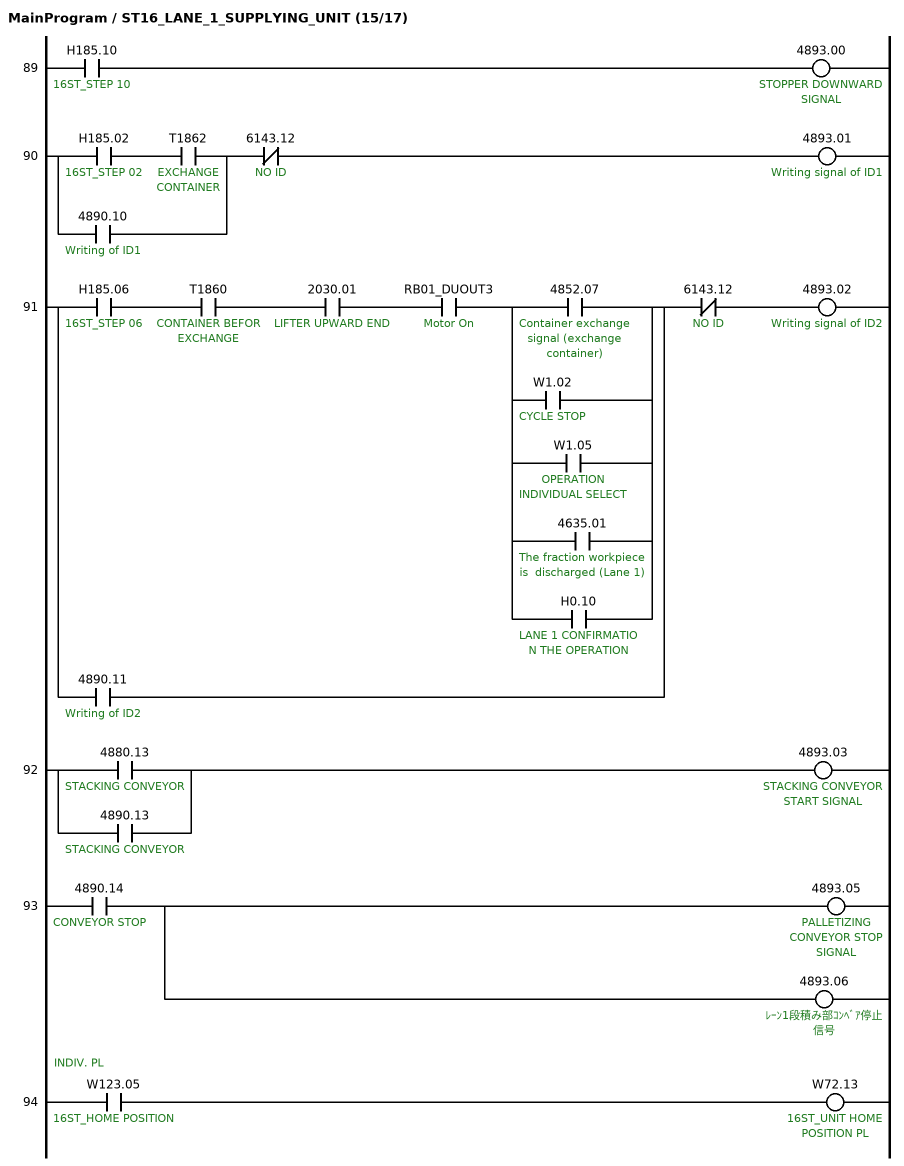
; [picture p648: MainProgram / ST16_LANE_1_SUPPLYING_UNIT, rungs 89-94]
; rung 89
LD H185.10  ; 16ST_STEP 10
OUT 4893.00  ; STOPPER DOWNWARD SIGNAL
; rung 90
LD H185.02  ; 16ST_STEP 02
AND T1862  ; EXCHANGE CONTAINER
OR 4890.10  ; Writing of ID1
ANDNOT 6143.12  ; NO ID
OUT 4893.01  ; Writing signal of ID1
; rung 91
LD H185.06  ; 16ST_STEP 06
AND T1860  ; CONTAINER BEFOR EXCHANGE
AND 2030.01  ; LIFTER UPWARD END
AND RB01_DUOUT3  ; Motor On
LD 4852.07  ; Container exchange signal (exchange container)
OR W1.02  ; CYCLE STOP
OR W1.05  ; OPERATION INDIVIDUAL SELECT
OR 4635.01  ; The fraction workpiece is  discharged (Lane 1)
OR H0.10  ; LANE 1 CONFIRMATION THE OPERATION
ANDLD
OR 4890.11  ; Writing of ID2
ANDNOT 6143.12  ; NO ID
OUT 4893.02  ; Writing signal of ID2
; rung 92
LD 4880.13  ; STACKING CONVEYOR
OR 4890.13  ; STACKING CONVEYOR
OUT 4893.03  ; STACKING CONVEYOR START SIGNAL
; rung 93
LD 4890.14  ; CONVEYOR STOP
OUT 4893.05  ; PALLETIZING CONVEYOR STOP SIGNAL
OUT 4893.06  ; ﾚｰﾝ1段積み部ｺﾝﾍﾞｱ停止信号
; rung 94: INDIV. PL
LD W123.05  ; 16ST_HOME POSITION
OUT W72.13  ; 16ST_UNIT HOME POSITION PL

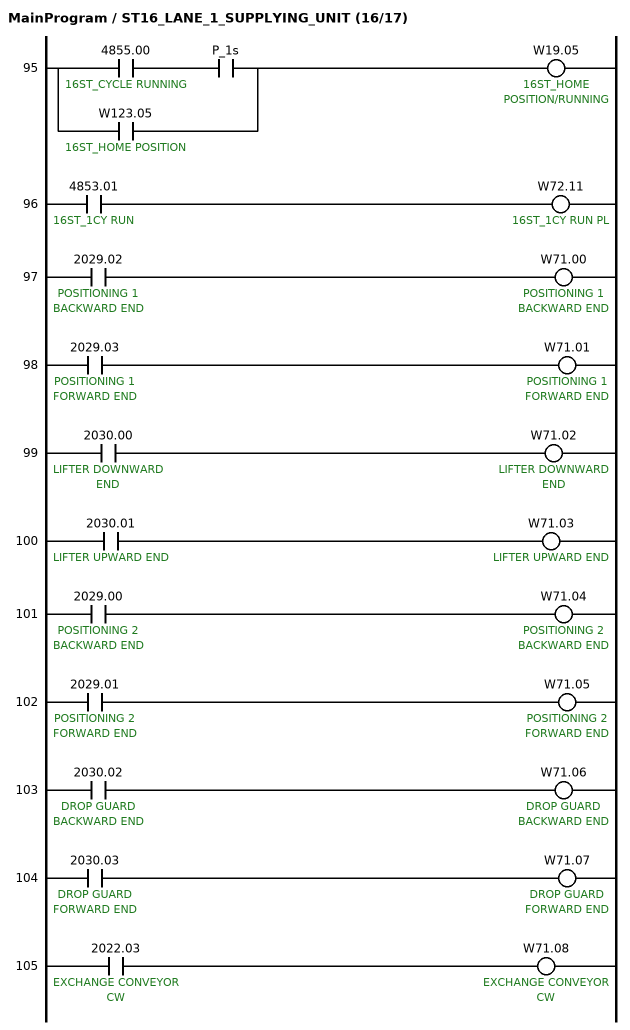
; rung 95
LD 4855.00  ; 16ST_CYCLE RUNNING
AND P_1s
OR W123.05  ; 16ST_HOME POSITION
OUT W19.05  ; 16ST_HOME POSITION/RUNNING
; rung 96
LD 4853.01  ; 16ST_1CY RUN
OUT W72.11  ; 16ST_1CY RUN PL
; rung 97
LD 2029.02  ; POSITIONING 1 BACKWARD END
OUT W71.00  ; POSITIONING 1 BACKWARD END
; rung 98
LD 2029.03  ; POSITIONING 1 FORWARD END
OUT W71.01  ; POSITIONING 1 FORWARD END
; rung 99
LD 2030.00  ; LIFTER DOWNWARD END
OUT W71.02  ; LIFTER DOWNWARD END
; rung 100
LD 2030.01  ; LIFTER UPWARD END
OUT W71.03  ; LIFTER UPWARD END
; rung 101
LD 2029.00  ; POSITIONING 2 BACKWARD END
OUT W71.04  ; POSITIONING 2 BACKWARD END
; rung 102
LD 2029.01  ; POSITIONING 2 FORWARD END
OUT W71.05  ; POSITIONING 2 FORWARD END
; rung 103
LD 2030.02  ; DROP GUARD BACKWARD END
OUT W71.06  ; DROP GUARD BACKWARD END
; rung 104
LD 2030.03  ; DROP GUARD FORWARD END
OUT W71.07  ; DROP GUARD FORWARD END
; rung 105
LD 2022.03  ; EXCHANGE CONVEYOR CW
OUT W71.08  ; EXCHANGE CONVEYOR CW

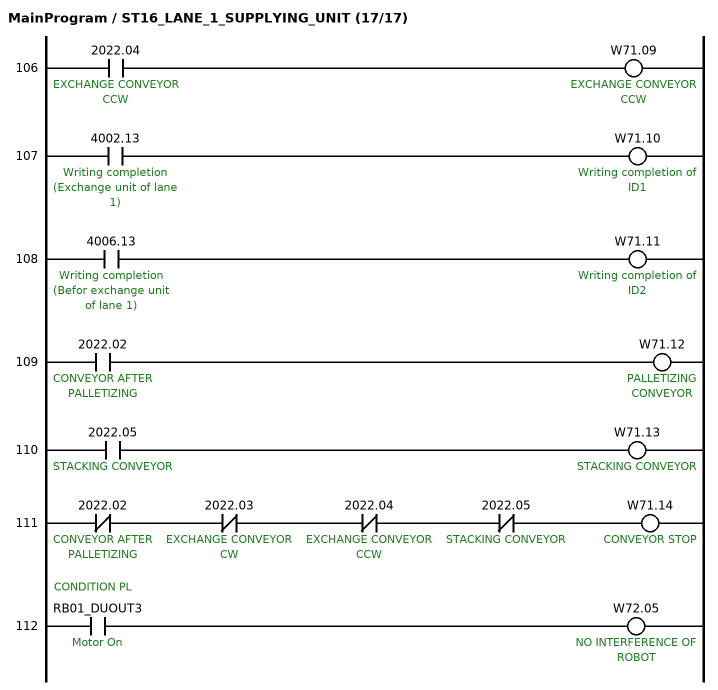
; rung 106
LD 2022.04  ; EXCHANGE CONVEYOR CCW
OUT W71.09  ; EXCHANGE CONVEYOR CCW
; rung 107
LD 4002.13  ; Writing completion (Exchange unit of lane 1)
OUT W71.10  ; Writing completion of ID1
; rung 108
LD 4006.13  ; Writing completion (Befor exchange unit of lane 1)
OUT W71.11  ; Writing completion of ID2
; rung 109
LD 2022.02  ; CONVEYOR AFTER PALLETIZING
OUT W71.12  ; PALLETIZING CONVEYOR
; rung 110
LD 2022.05  ; STACKING CONVEYOR
OUT W71.13  ; STACKING CONVEYOR
; rung 111
LDNOT 2022.02  ; CONVEYOR AFTER PALLETIZING
ANDNOT 2022.03  ; EXCHANGE CONVEYOR CW
ANDNOT 2022.04  ; EXCHANGE CONVEYOR CCW
ANDNOT 2022.05  ; STACKING CONVEYOR
OUT W71.14  ; CONVEYOR STOP
; rung 112: CONDITION PL
LD RB01_DUOUT3  ; Motor On
OUT W72.05  ; NO INTERFERENCE OF ROBOT

### Section ST17_LANE_1_STACKING_UNIT

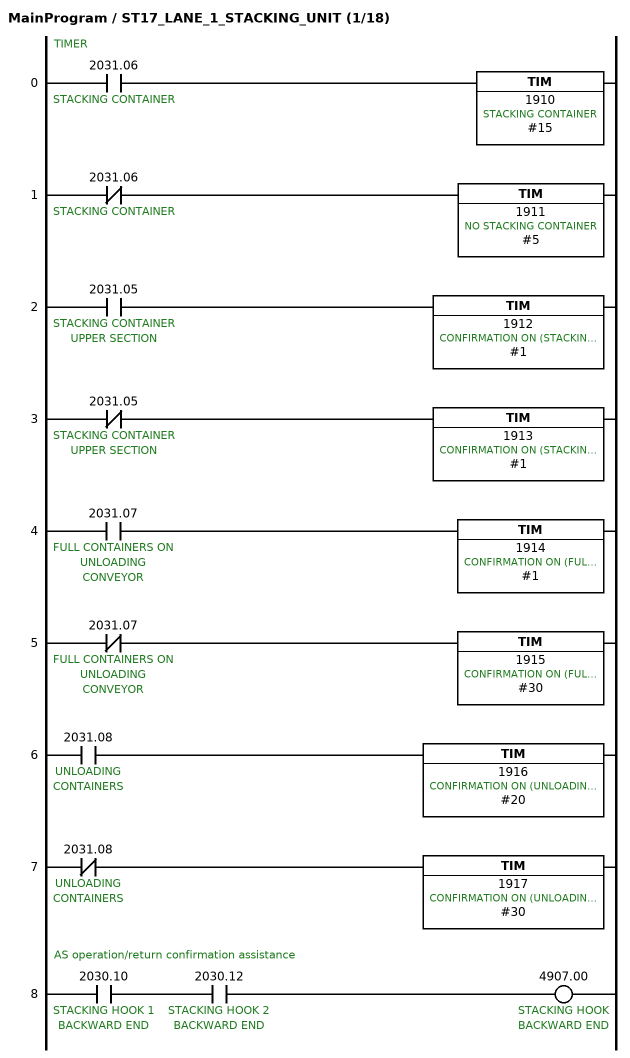
; rung 0: TIMER
LD 2031.06  ; STACKING CONTAINER
TIM 1910 #15  ; STACKING CONTAINER
; rung 1
LDNOT 2031.06  ; STACKING CONTAINER
TIM 1911 #5  ; NO STACKING CONTAINER
; rung 2
LD 2031.05  ; STACKING CONTAINER UPPER SECTION
TIM 1912 #1  ; CONFIRMATION ON (STACKING CONTAINER UPPER SECTION)
; rung 3
LDNOT 2031.05  ; STACKING CONTAINER UPPER SECTION
TIM 1913 #1  ; CONFIRMATION ON (STACKING CONTAINER UPPER SECTION)
; rung 4
LD 2031.07  ; FULL CONTAINERS ON UNLOADING CONVEYOR
TIM 1914 #1  ; CONFIRMATION ON (FULL CONTAINERS ON UNLOADING CONVEYOR)
; rung 5
LDNOT 2031.07  ; FULL CONTAINERS ON UNLOADING CONVEYOR
TIM 1915 #30  ; CONFIRMATION ON (FULL CONTAINERS ON UNLOADING CONVEYOR)
; rung 6
LD 2031.08  ; UNLOADING CONTAINERS
TIM 1916 #20  ; CONFIRMATION ON (UNLOADING CONTAINERS)
; rung 7
LDNOT 2031.08  ; UNLOADING CONTAINERS
TIM 1917 #30  ; CONFIRMATION ON (UNLOADING CONTAINERS)
; rung 8: AS operation/return confirmation assistance
LD 2030.10  ; STACKING HOOK 1 BACKWARD END
AND 2030.12  ; STACKING HOOK 2 BACKWARD END
OUT 4907.00  ; STACKING HOOK BACKWARD END

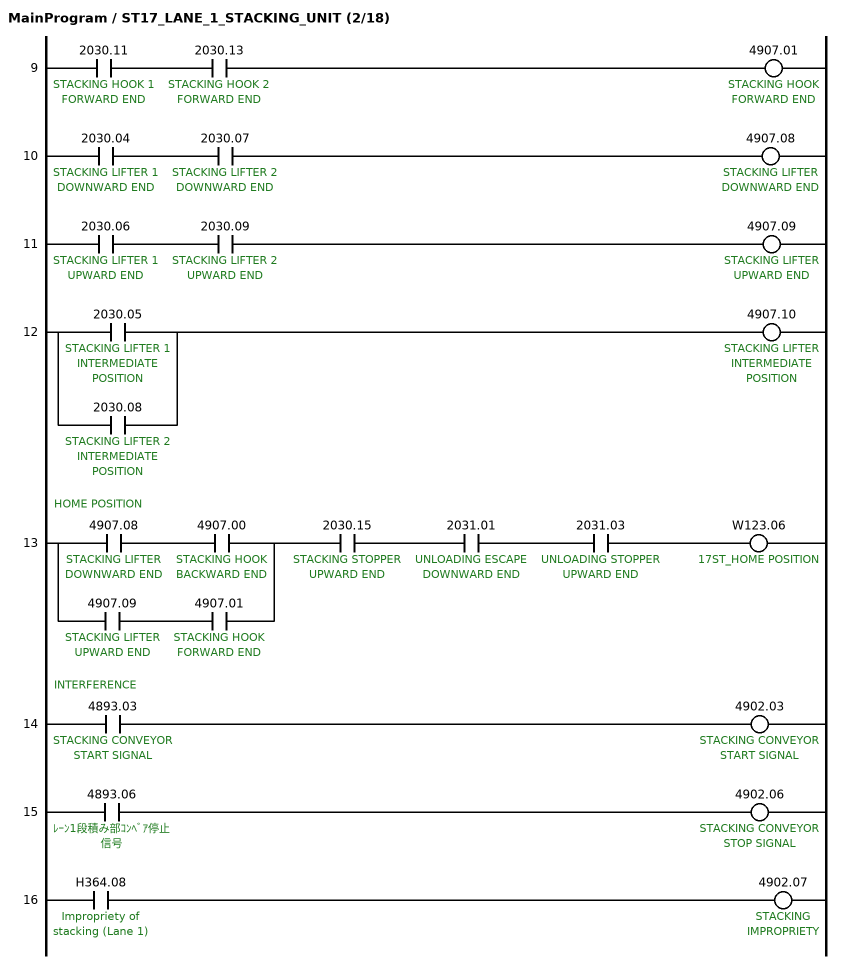
; rung 9
LD 2030.11  ; STACKING HOOK 1 FORWARD END
AND 2030.13  ; STACKING HOOK 2 FORWARD END
OUT 4907.01  ; STACKING HOOK FORWARD END
; rung 10
LD 2030.04  ; STACKING LIFTER 1 DOWNWARD END
AND 2030.07  ; STACKING LIFTER 2 DOWNWARD END
OUT 4907.08  ; STACKING LIFTER DOWNWARD END
; rung 11
LD 2030.06  ; STACKING LIFTER 1 UPWARD END
AND 2030.09  ; STACKING LIFTER 2 UPWARD END
OUT 4907.09  ; STACKING LIFTER UPWARD END
; rung 12
LD 2030.05  ; STACKING LIFTER 1 INTERMEDIATE POSITION
OR 2030.08  ; STACKING LIFTER 2 INTERMEDIATE POSITION
OUT 4907.10  ; STACKING LIFTER INTERMEDIATE POSITION
; rung 13: HOME POSITION
LD 4907.08  ; STACKING LIFTER DOWNWARD END
AND 4907.00  ; STACKING HOOK BACKWARD END
LD 4907.09  ; STACKING LIFTER UPWARD END
AND 4907.01  ; STACKING HOOK FORWARD END
ORLD
AND 2030.15  ; STACKING STOPPER UPWARD END
AND 2031.01  ; UNLOADING ESCAPE DOWNWARD END
AND 2031.03  ; UNLOADING STOPPER UPWARD END
OUT W123.06  ; 17ST_HOME POSITION
; rung 14: INTERFERENCE
LD 4893.03  ; STACKING CONVEYOR START SIGNAL
OUT 4902.03  ; STACKING CONVEYOR START SIGNAL
; rung 15
LD 4893.06  ; ﾚｰﾝ1段積み部ｺﾝﾍﾞｱ停止信号
OUT 4902.06  ; STACKING CONVEYOR STOP SIGNAL
; rung 16
LD H364.08  ; Impropriety of stacking (Lane 1)
OUT 4902.07  ; STACKING IMPROPRIETY

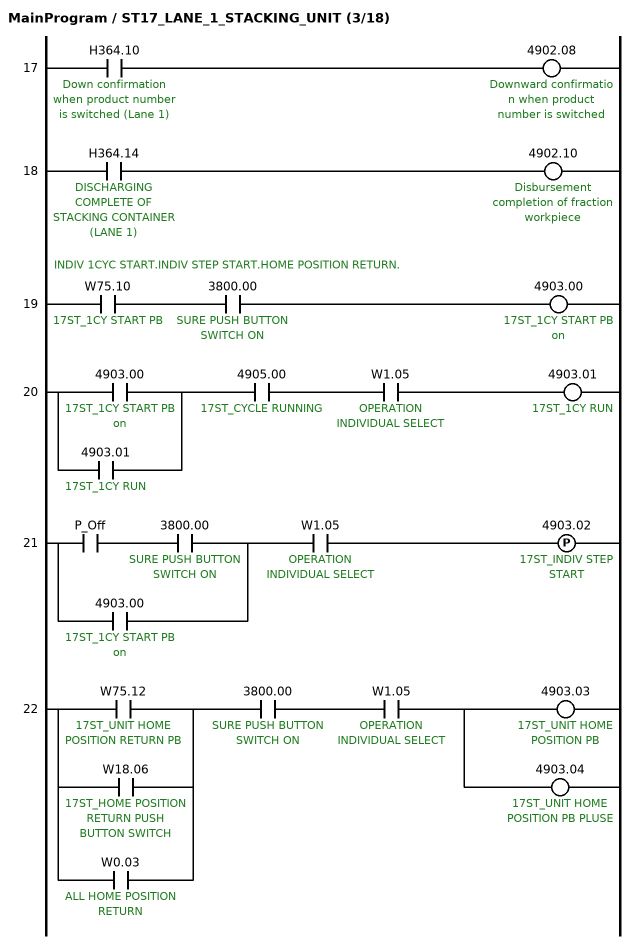
; rung 17
LD H364.10  ; Down confirmation when product number is switched (Lane 1)
OUT 4902.08  ; Downward confirmation when product number is switched
; rung 18
LD H364.14  ; DISCHARGING COMPLETE OF STACKING CONTAINER  (LANE 1)
OUT 4902.10  ; Disbursement completion of fraction workpiece
; rung 19: INDIV 1CYC START.INDIV STEP START.HOME POSITION RETURN.
LD W75.10  ; 17ST_1CY START PB
AND 3800.00  ; SURE PUSH BUTTON SWITCH ON
OUT 4903.00  ; 17ST_1CY START PB on
; rung 20
LD 4903.00  ; 17ST_1CY START PB on
OR 4903.01  ; 17ST_1CY RUN
AND 4905.00  ; 17ST_CYCLE RUNNING
AND W1.05  ; OPERATION INDIVIDUAL SELECT
OUT 4903.01  ; 17ST_1CY RUN
; rung 21
LD P_Off
AND 3800.00  ; SURE PUSH BUTTON SWITCH ON
OR 4903.00  ; 17ST_1CY START PB on
AND W1.05  ; OPERATION INDIVIDUAL SELECT
DIFU(013) 4903.02  ; 17ST_INDIV STEP START
; rung 22
LD W75.12  ; 17ST_UNIT HOME POSITION RETURN PB
OR W18.06  ; 17ST_HOME POSITION RETURN PUSH BUTTON SWITCH
OR W0.03  ; ALL HOME POSITION RETURN
AND 3800.00  ; SURE PUSH BUTTON SWITCH ON
AND W1.05  ; OPERATION INDIVIDUAL SELECT
OUT 4903.03  ; 17ST_UNIT HOME POSITION PB
OUT 4903.04  ; 17ST_UNIT HOME POSITION PB PLUSE

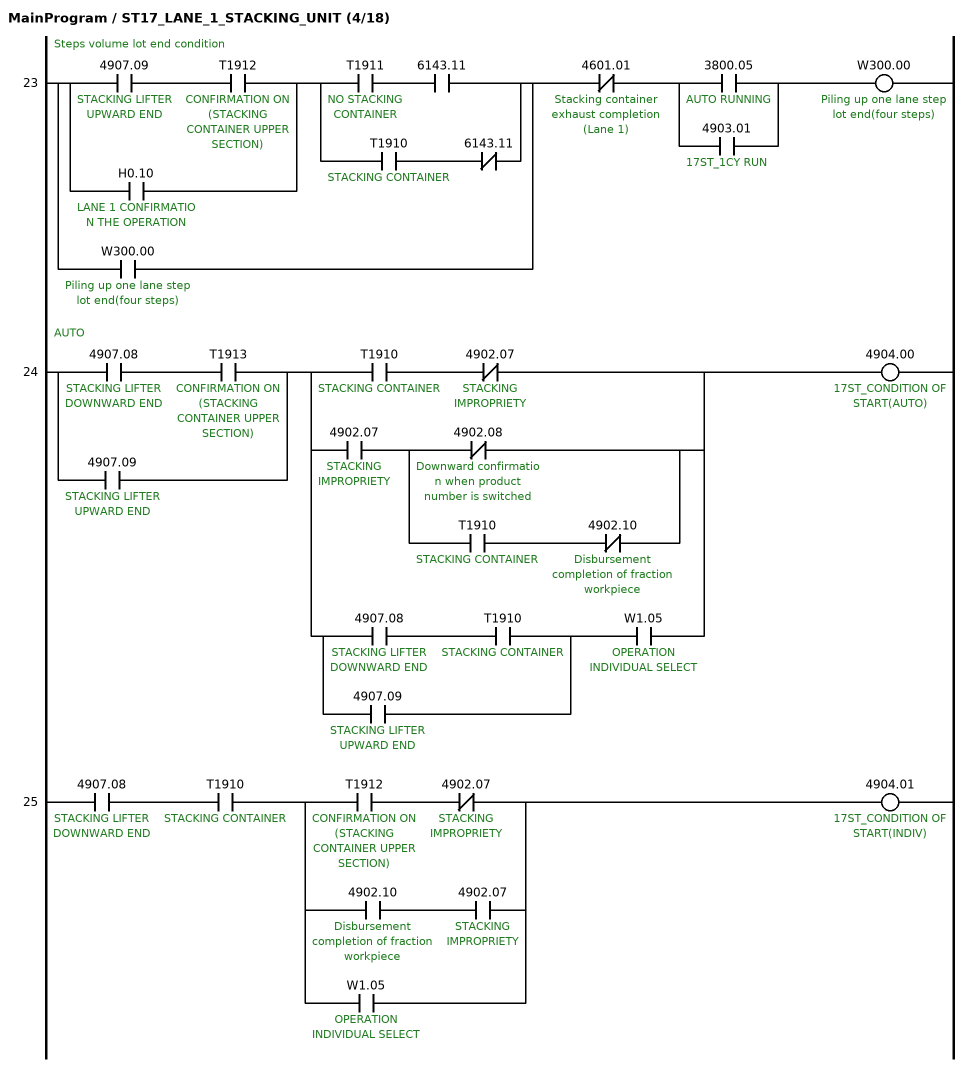
; rung 23: Steps volume lot end condition
LD 4907.09  ; STACKING LIFTER UPWARD END
AND T1912  ; CONFIRMATION ON (STACKING CONTAINER UPPER SECTION)
OR H0.10  ; LANE 1 CONFIRMATION THE OPERATION
LD T1911  ; NO STACKING CONTAINER
AND 6143.11
LD T1910  ; STACKING CONTAINER
ANDNOT 6143.11
ORLD
ANDLD
OR W300.00  ; Piling up one lane step lot end(four steps)
ANDNOT 4601.01  ; Stacking container exhaust completion (Lane 1)
LD 3800.05  ; AUTO RUNNING
OR 4903.01  ; 17ST_1CY RUN
ANDLD
OUT W300.00  ; Piling up one lane step lot end(four steps)
; rung 24: AUTO
LD 4907.08  ; STACKING LIFTER DOWNWARD END
AND T1913  ; CONFIRMATION ON (STACKING CONTAINER UPPER SECTION)
OR 4907.09  ; STACKING LIFTER UPWARD END
LD T1910  ; STACKING CONTAINER
ANDNOT 4902.07  ; STACKING IMPROPRIETY
LD 4902.07  ; STACKING IMPROPRIETY
LDNOT 4902.08  ; Downward confirmation when product number is switched
LD T1910  ; STACKING CONTAINER
ANDNOT 4902.10  ; Disbursement completion of fraction workpiece
ORLD
ANDLD
ORLD
LD 4907.08  ; STACKING LIFTER DOWNWARD END
AND T1910  ; STACKING CONTAINER
OR 4907.09  ; STACKING LIFTER UPWARD END
AND W1.05  ; OPERATION INDIVIDUAL SELECT
ORLD
ANDLD
OUT 4904.00  ; 17ST_CONDITION OF START(AUTO)
; rung 25
LD 4907.08  ; STACKING LIFTER DOWNWARD END
AND T1910  ; STACKING CONTAINER
LD T1912  ; CONFIRMATION ON (STACKING CONTAINER UPPER SECTION)
ANDNOT 4902.07  ; STACKING IMPROPRIETY
LD 4902.10  ; Disbursement completion of fraction workpiece
AND 4902.07  ; STACKING IMPROPRIETY
ORLD
OR W1.05  ; OPERATION INDIVIDUAL SELECT
ANDLD
OUT 4904.01  ; 17ST_CONDITION OF START(INDIV)

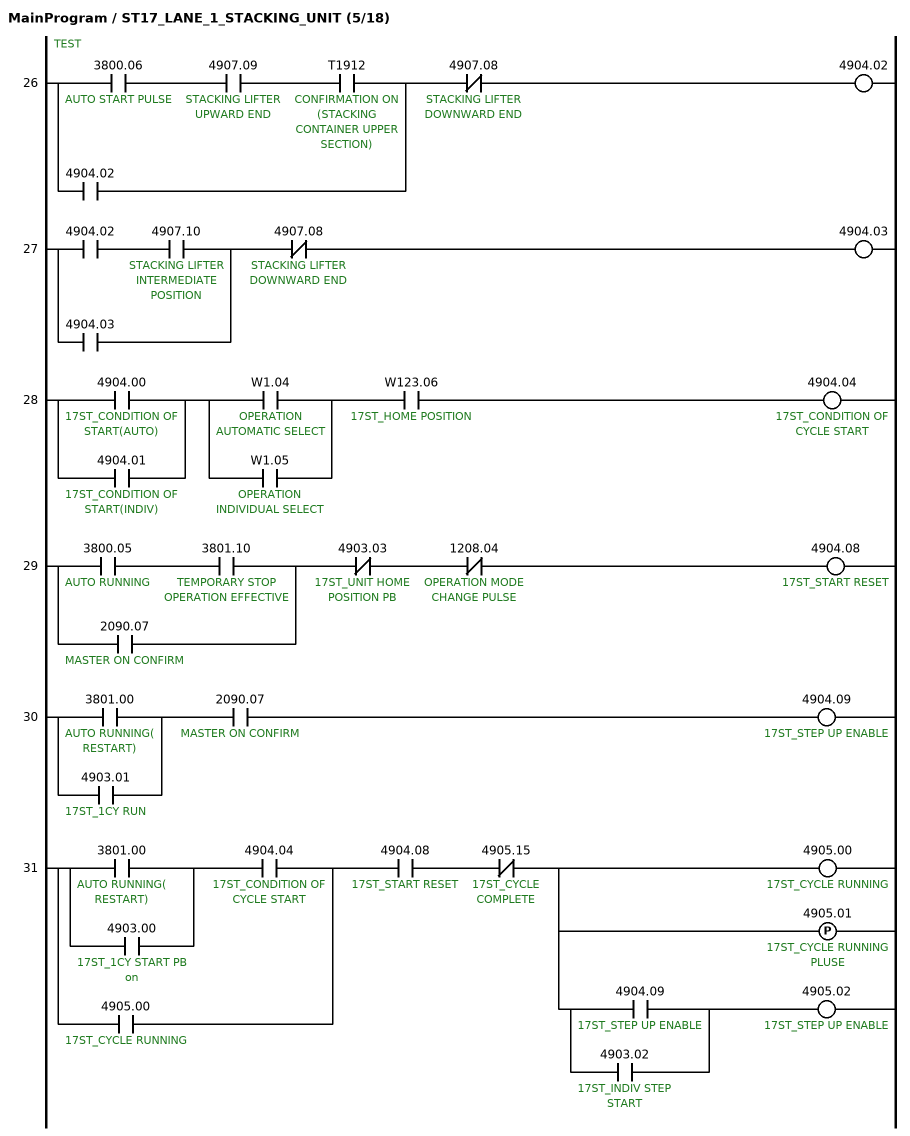
; rung 26: TEST
LD 3800.06  ; AUTO START PULSE
AND 4907.09  ; STACKING LIFTER UPWARD END
AND T1912  ; CONFIRMATION ON (STACKING CONTAINER UPPER SECTION)
OR 4904.02
ANDNOT 4907.08  ; STACKING LIFTER DOWNWARD END
OUT 4904.02
; rung 27
LD 4904.02
AND 4907.10  ; STACKING LIFTER INTERMEDIATE POSITION
OR 4904.03
ANDNOT 4907.08  ; STACKING LIFTER DOWNWARD END
OUT 4904.03
; rung 28
LD 4904.00  ; 17ST_CONDITION OF START(AUTO)
OR 4904.01  ; 17ST_CONDITION OF START(INDIV)
LD W1.04  ; OPERATION AUTOMATIC SELECT
OR W1.05  ; OPERATION INDIVIDUAL SELECT
ANDLD
AND W123.06  ; 17ST_HOME POSITION
OUT 4904.04  ; 17ST_CONDITION OF CYCLE START
; rung 29
LD 3800.05  ; AUTO RUNNING
AND 3801.10  ; TEMPORARY STOP OPERATION EFFECTIVE
OR 2090.07  ; MASTER ON CONFIRM
ANDNOT 4903.03  ; 17ST_UNIT HOME POSITION PB
ANDNOT 1208.04  ; OPERATION MODE CHANGE PULSE
OUT 4904.08  ; 17ST_START RESET
; rung 30
LD 3801.00  ; AUTO RUNNING(RESTART)
OR 4903.01  ; 17ST_1CY RUN
AND 2090.07  ; MASTER ON CONFIRM
OUT 4904.09  ; 17ST_STEP UP ENABLE
; rung 31
LD 3801.00  ; AUTO RUNNING(RESTART)
OR 4903.00  ; 17ST_1CY START PB on
AND 4904.04  ; 17ST_CONDITION OF CYCLE START
OR 4905.00  ; 17ST_CYCLE RUNNING
AND 4904.08  ; 17ST_START RESET
ANDNOT 4905.15  ; 17ST_CYCLE COMPLETE
OUT 4905.00  ; 17ST_CYCLE RUNNING
DIFU(013) 4905.01  ; 17ST_CYCLE RUNNING PLUSE
LD 4904.09  ; 17ST_STEP UP ENABLE
OR 4903.02  ; 17ST_INDIV STEP START
ANDLD
OUT 4905.02  ; 17ST_STEP UP ENABLE

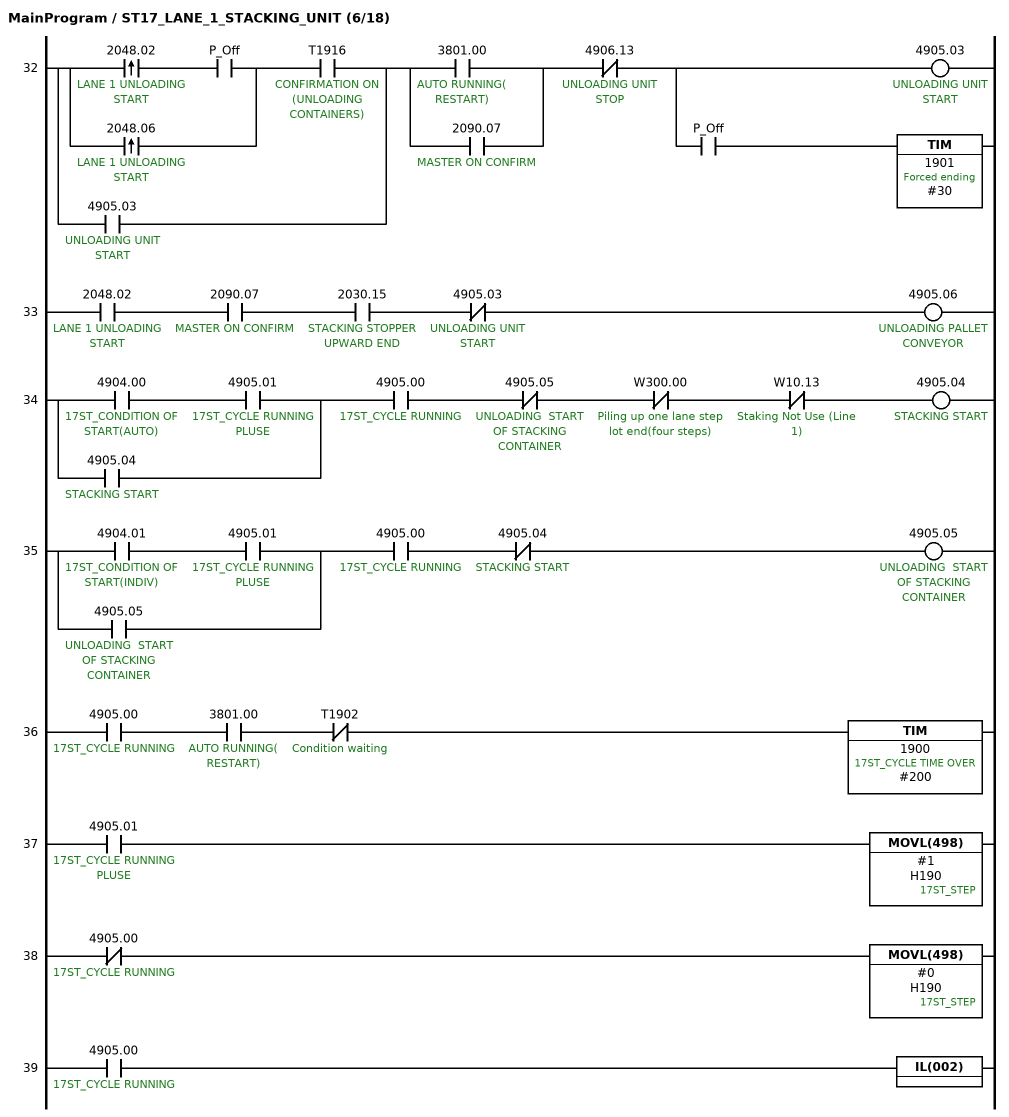
; rung 32
@LD 2048.02  ; LANE 1 UNLOADING START
AND P_Off
@OR 2048.06  ; LANE 1 UNLOADING START
AND T1916  ; CONFIRMATION ON (UNLOADING CONTAINERS)
OR 4905.03  ; UNLOADING UNIT START
LD 3801.00  ; AUTO RUNNING(RESTART)
OR 2090.07  ; MASTER ON CONFIRM
ANDLD
ANDNOT 4906.13  ; UNLOADING UNIT STOP
OUT 4905.03  ; UNLOADING UNIT START
AND P_Off
TIM 1901 #30  ; Forced ending
; rung 33
LD 2048.02  ; LANE 1 UNLOADING START
AND 2090.07  ; MASTER ON CONFIRM
AND 2030.15  ; STACKING STOPPER UPWARD END
ANDNOT 4905.03  ; UNLOADING UNIT START
OUT 4905.06  ; UNLOADING PALLET CONVEYOR
; rung 34
LD 4904.00  ; 17ST_CONDITION OF START(AUTO)
AND 4905.01  ; 17ST_CYCLE RUNNING PLUSE
OR 4905.04  ; STACKING START
AND 4905.00  ; 17ST_CYCLE RUNNING
ANDNOT 4905.05  ; UNLOADING  START OF STACKING CONTAINER
ANDNOT W300.00  ; Piling up one lane step lot end(four steps)
ANDNOT W10.13  ; Staking Not Use (Line 1)
OUT 4905.04  ; STACKING START
; rung 35
LD 4904.01  ; 17ST_CONDITION OF START(INDIV)
AND 4905.01  ; 17ST_CYCLE RUNNING PLUSE
OR 4905.05  ; UNLOADING  START OF STACKING CONTAINER
AND 4905.00  ; 17ST_CYCLE RUNNING
ANDNOT 4905.04  ; STACKING START
OUT 4905.05  ; UNLOADING  START OF STACKING CONTAINER
; rung 36
LD 4905.00  ; 17ST_CYCLE RUNNING
AND 3801.00  ; AUTO RUNNING(RESTART)
ANDNOT T1902  ; Condition waiting
TIM 1900 #200  ; 17ST_CYCLE TIME OVER
; rung 37
LD 4905.01  ; 17ST_CYCLE RUNNING PLUSE
MOVL(498) #1 H190  ; 17ST_STEP
; rung 38
LDNOT 4905.00  ; 17ST_CYCLE RUNNING
MOVL(498) #0 H190  ; 17ST_STEP
; rung 39
LD 4905.00  ; 17ST_CYCLE RUNNING
IL(002)

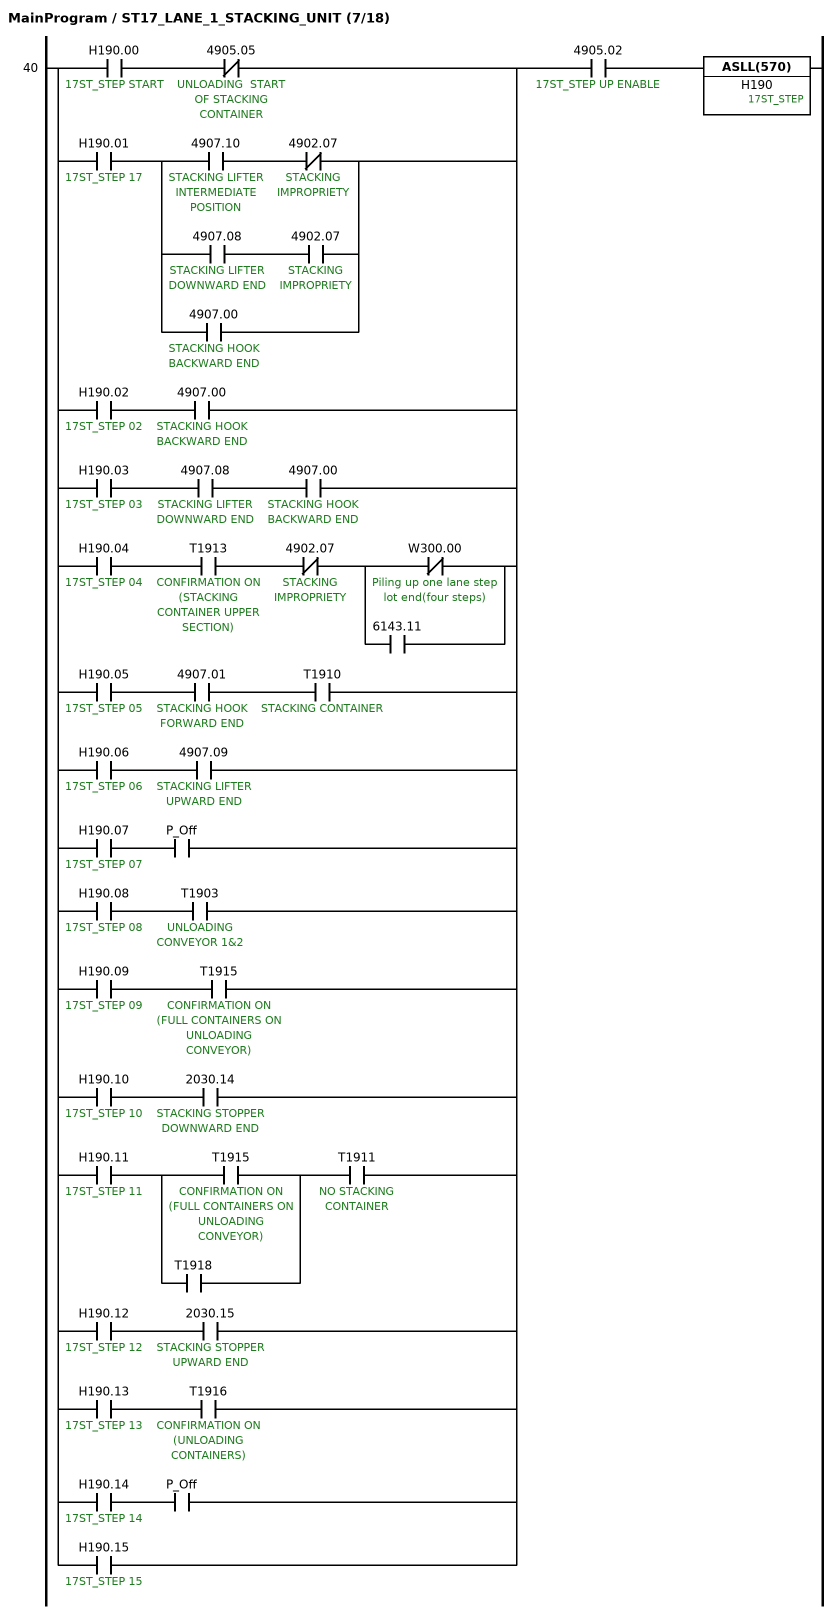
; rung 40
LD H190.00  ; 17ST_STEP START
ANDNOT 4905.05  ; UNLOADING  START OF STACKING CONTAINER
LD H190.01  ; 17ST_STEP 17
LD 4907.10  ; STACKING LIFTER INTERMEDIATE POSITION
ANDNOT 4902.07  ; STACKING IMPROPRIETY
LD 4907.08  ; STACKING LIFTER DOWNWARD END
AND 4902.07  ; STACKING IMPROPRIETY
ORLD
OR 4907.00  ; STACKING HOOK BACKWARD END
ANDLD
ORLD
LD H190.02  ; 17ST_STEP 02
AND 4907.00  ; STACKING HOOK BACKWARD END
ORLD
LD H190.03  ; 17ST_STEP 03
AND 4907.08  ; STACKING LIFTER DOWNWARD END
AND 4907.00  ; STACKING HOOK BACKWARD END
ORLD
LD H190.04  ; 17ST_STEP 04
AND T1913  ; CONFIRMATION ON (STACKING CONTAINER UPPER SECTION)
ANDNOT 4902.07  ; STACKING IMPROPRIETY
LDNOT W300.00  ; Piling up one lane step lot end(four steps)
OR 6143.11
ANDLD
ORLD
LD H190.05  ; 17ST_STEP 05
AND 4907.01  ; STACKING HOOK FORWARD END
AND T1910  ; STACKING CONTAINER
ORLD
LD H190.06  ; 17ST_STEP 06
AND 4907.09  ; STACKING LIFTER UPWARD END
ORLD
LD H190.07  ; 17ST_STEP 07
AND P_Off
ORLD
LD H190.08  ; 17ST_STEP 08
AND T1903  ; UNLOADING CONVEYOR 1&2
ORLD
LD H190.09  ; 17ST_STEP 09
AND T1915  ; CONFIRMATION ON (FULL CONTAINERS ON UNLOADING CONVEYOR)
ORLD
LD H190.10  ; 17ST_STEP 10
AND 2030.14  ; STACKING STOPPER DOWNWARD END
ORLD
LD H190.11  ; 17ST_STEP 11
LD T1915  ; CONFIRMATION ON (FULL CONTAINERS ON UNLOADING CONVEYOR)
OR T1918
ANDLD
AND T1911  ; NO STACKING CONTAINER
ORLD
LD H190.12  ; 17ST_STEP 12
AND 2030.15  ; STACKING STOPPER UPWARD END
ORLD
LD H190.13  ; 17ST_STEP 13
AND T1916  ; CONFIRMATION ON (UNLOADING CONTAINERS)
ORLD
LD H190.14  ; 17ST_STEP 14
AND P_Off
ORLD
OR H190.15  ; 17ST_STEP 15
AND 4905.02  ; 17ST_STEP UP ENABLE
ASLL(570) H190  ; 17ST_STEP

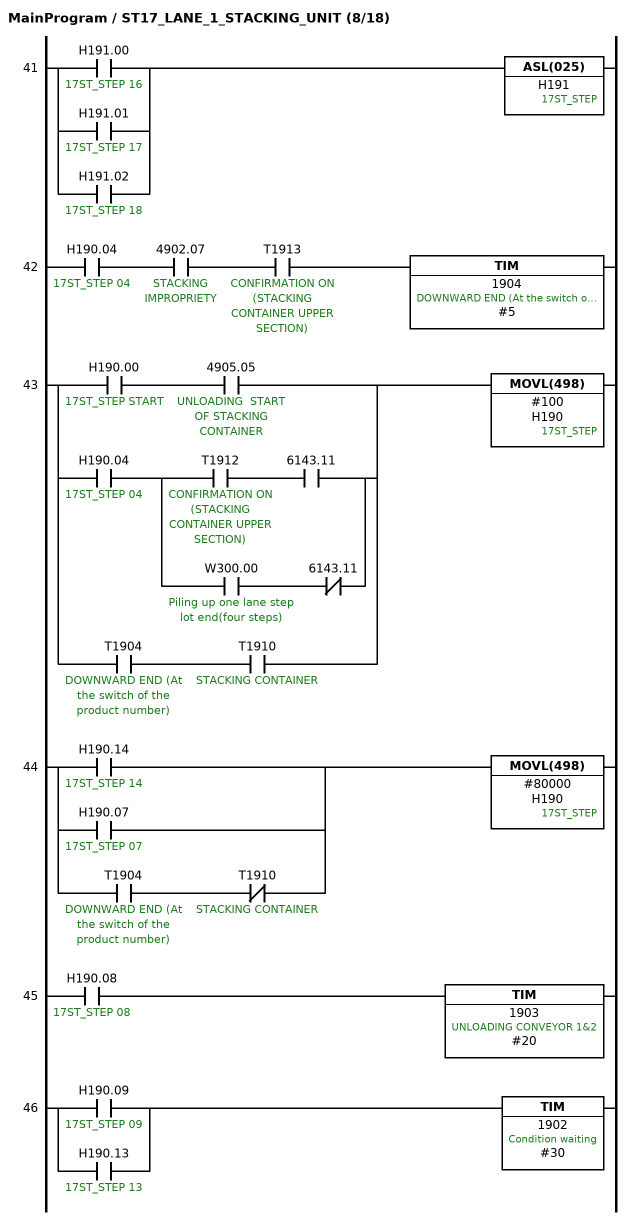
; rung 41
LD H191.00  ; 17ST_STEP 16
OR H191.01  ; 17ST_STEP 17
OR H191.02  ; 17ST_STEP 18
ASL(025) H191  ; 17ST_STEP
; rung 42
LD H190.04  ; 17ST_STEP 04
AND 4902.07  ; STACKING IMPROPRIETY
AND T1913  ; CONFIRMATION ON (STACKING CONTAINER UPPER SECTION)
TIM 1904 #5  ; DOWNWARD END (At the switch of the product number)
; rung 43
LD H190.00  ; 17ST_STEP START
AND 4905.05  ; UNLOADING  START OF STACKING CONTAINER
LD H190.04  ; 17ST_STEP 04
LD T1912  ; CONFIRMATION ON (STACKING CONTAINER UPPER SECTION)
AND 6143.11
LD W300.00  ; Piling up one lane step lot end(four steps)
ANDNOT 6143.11
ORLD
ANDLD
ORLD
LD T1904  ; DOWNWARD END (At the switch of the product number)
AND T1910  ; STACKING CONTAINER
ORLD
MOVL(498) #100 H190  ; 17ST_STEP
; rung 44
LD H190.14  ; 17ST_STEP 14
OR H190.07  ; 17ST_STEP 07
LD T1904  ; DOWNWARD END (At the switch of the product number)
ANDNOT T1910  ; STACKING CONTAINER
ORLD
MOVL(498) #80000 H190  ; 17ST_STEP
; rung 45
LD H190.08  ; 17ST_STEP 08
TIM 1903 #20  ; UNLOADING CONVEYOR 1&2
; rung 46
LD H190.09  ; 17ST_STEP 09
OR H190.13  ; 17ST_STEP 13
TIM 1902 #30  ; Condition waiting

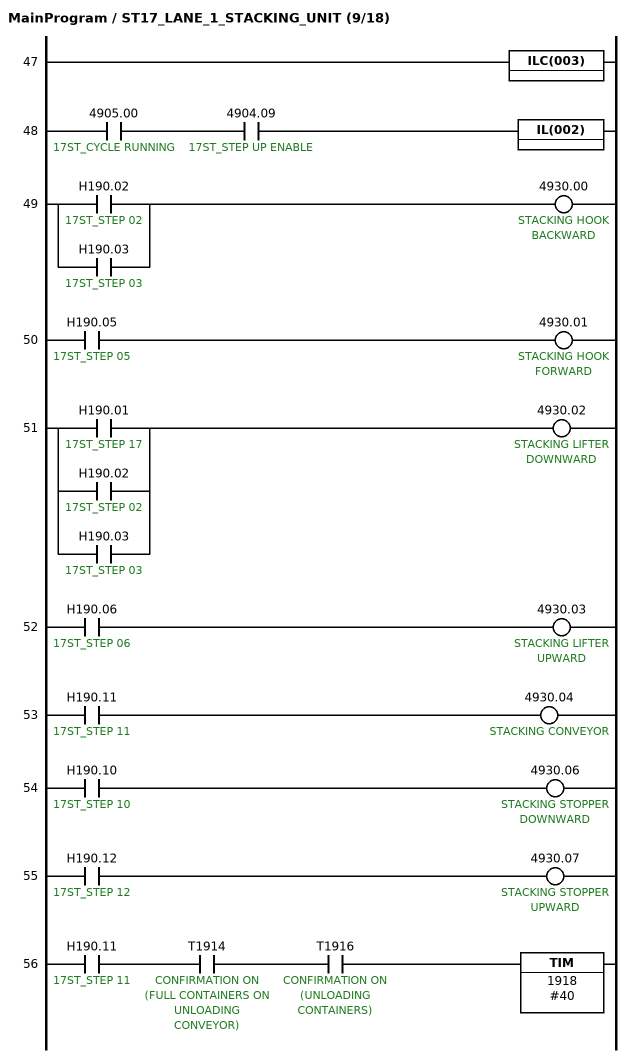
; rung 47
ILC(003)
; rung 48
LD 4905.00  ; 17ST_CYCLE RUNNING
AND 4904.09  ; 17ST_STEP UP ENABLE
IL(002)
; rung 49
LD H190.02  ; 17ST_STEP 02
OR H190.03  ; 17ST_STEP 03
OUT 4930.00  ; STACKING HOOK BACKWARD
; rung 50
LD H190.05  ; 17ST_STEP 05
OUT 4930.01  ; STACKING HOOK FORWARD
; rung 51
LD H190.01  ; 17ST_STEP 17
OR H190.02  ; 17ST_STEP 02
OR H190.03  ; 17ST_STEP 03
OUT 4930.02  ; STACKING LIFTER DOWNWARD
; rung 52
LD H190.06  ; 17ST_STEP 06
OUT 4930.03  ; STACKING LIFTER UPWARD
; rung 53
LD H190.11  ; 17ST_STEP 11
OUT 4930.04  ; STACKING CONVEYOR
; rung 54
LD H190.10  ; 17ST_STEP 10
OUT 4930.06  ; STACKING STOPPER DOWNWARD
; rung 55
LD H190.12  ; 17ST_STEP 12
OUT 4930.07  ; STACKING STOPPER UPWARD
; rung 56
LD H190.11  ; 17ST_STEP 11
AND T1914  ; CONFIRMATION ON (FULL CONTAINERS ON UNLOADING CONVEYOR)
AND T1916  ; CONFIRMATION ON (UNLOADING CONTAINERS)
TIM 1918 #40

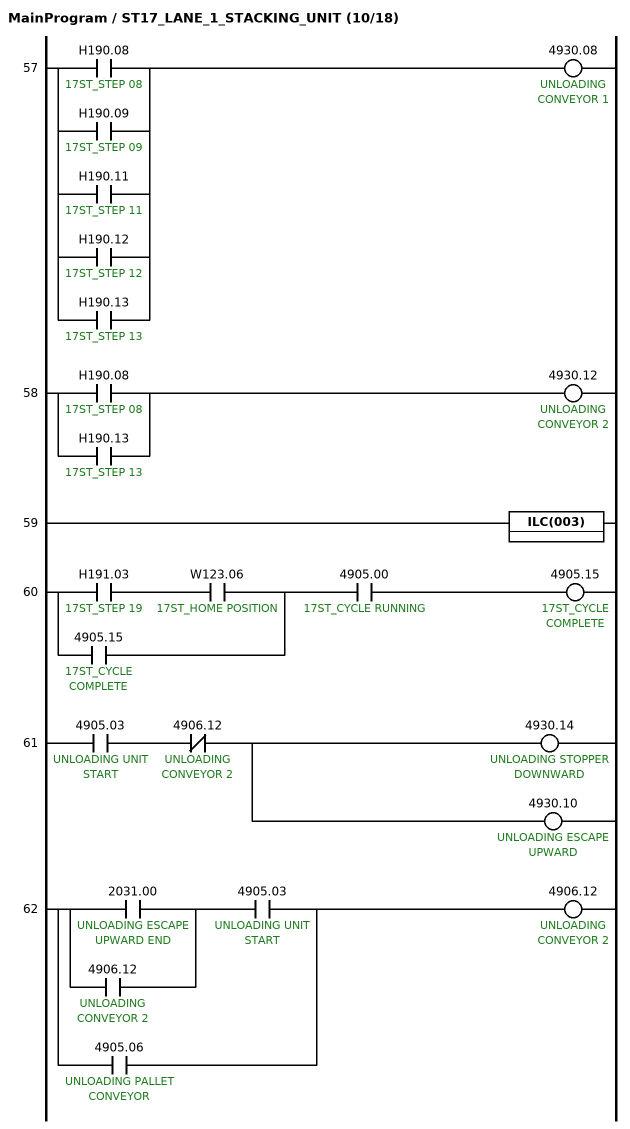
; rung 57
LD H190.08  ; 17ST_STEP 08
OR H190.09  ; 17ST_STEP 09
OR H190.11  ; 17ST_STEP 11
OR H190.12  ; 17ST_STEP 12
OR H190.13  ; 17ST_STEP 13
OUT 4930.08  ; UNLOADING CONVEYOR 1
; rung 58
LD H190.08  ; 17ST_STEP 08
OR H190.13  ; 17ST_STEP 13
OUT 4930.12  ; UNLOADING CONVEYOR 2
; rung 59
ILC(003)
; rung 60
LD H191.03  ; 17ST_STEP 19
AND W123.06  ; 17ST_HOME POSITION
OR 4905.15  ; 17ST_CYCLE COMPLETE
AND 4905.00  ; 17ST_CYCLE RUNNING
OUT 4905.15  ; 17ST_CYCLE COMPLETE
; rung 61
LD 4905.03  ; UNLOADING UNIT START
ANDNOT 4906.12  ; UNLOADING CONVEYOR 2
OUT 4930.14  ; UNLOADING STOPPER DOWNWARD
OUT 4930.10  ; UNLOADING ESCAPE UPWARD
; rung 62
LD 2031.00  ; UNLOADING ESCAPE UPWARD END
OR 4906.12  ; UNLOADING CONVEYOR 2
AND 4905.03  ; UNLOADING UNIT START
OR 4905.06  ; UNLOADING PALLET CONVEYOR
OUT 4906.12  ; UNLOADING CONVEYOR 2

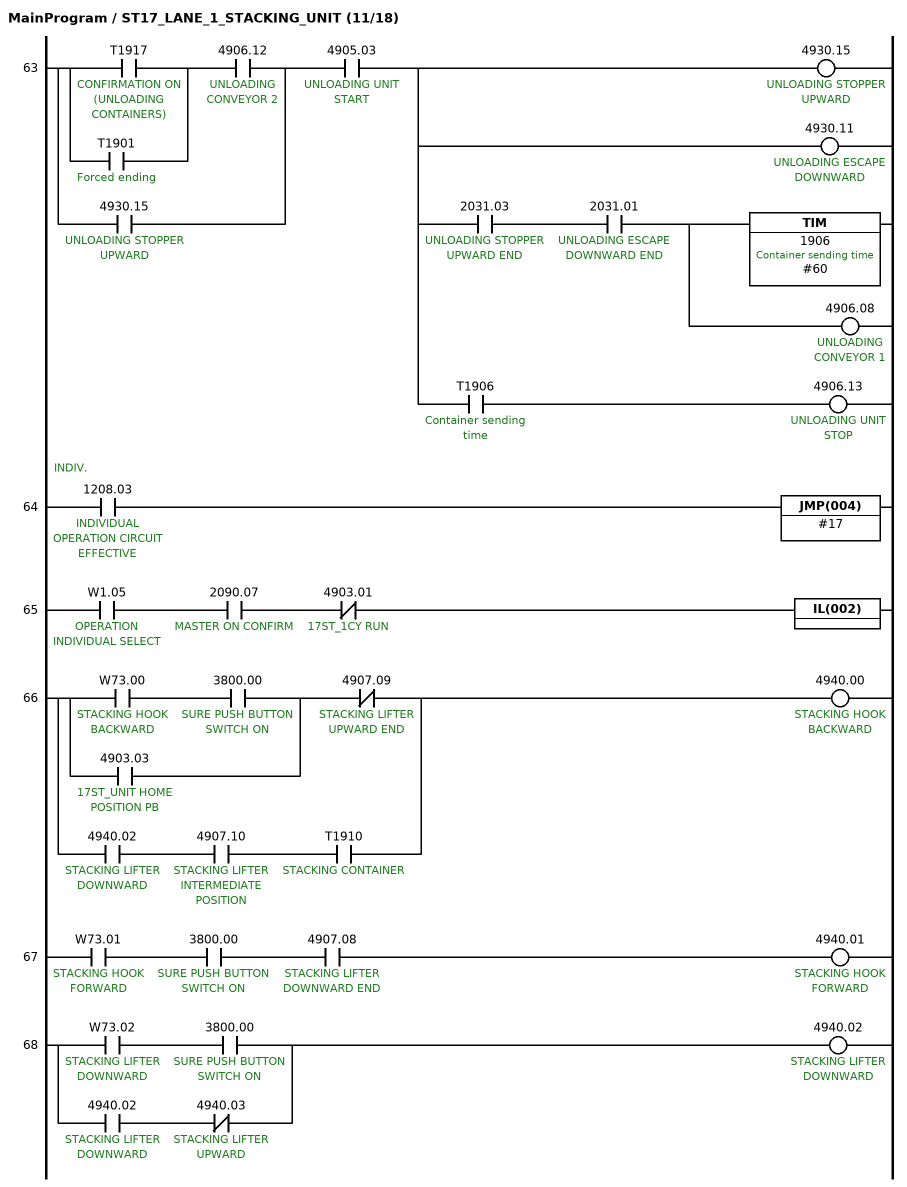
; rung 63
LD T1917  ; CONFIRMATION ON (UNLOADING CONTAINERS)
OR T1901  ; Forced ending
AND 4906.12  ; UNLOADING CONVEYOR 2
OR 4930.15  ; UNLOADING STOPPER UPWARD
AND 4905.03  ; UNLOADING UNIT START
OUT TR0
OUT 4930.15  ; UNLOADING STOPPER UPWARD
OUT 4930.11  ; UNLOADING ESCAPE DOWNWARD
AND 2031.03  ; UNLOADING STOPPER UPWARD END
AND 2031.01  ; UNLOADING ESCAPE DOWNWARD END
TIM 1906 #60  ; Container sending time
OUT 4906.08  ; UNLOADING CONVEYOR 1
LD TR0
AND T1906  ; Container sending time
OUT 4906.13  ; UNLOADING UNIT STOP
; rung 64: INDIV.
LD 1208.03  ; INDIVIDUAL OPERATION CIRCUIT EFFECTIVE
JMP(004) #17
; rung 65
LD W1.05  ; OPERATION INDIVIDUAL SELECT
AND 2090.07  ; MASTER ON CONFIRM
ANDNOT 4903.01  ; 17ST_1CY RUN
IL(002)
; rung 66
LD W73.00  ; STACKING HOOK BACKWARD
AND 3800.00  ; SURE PUSH BUTTON SWITCH ON
OR 4903.03  ; 17ST_UNIT HOME POSITION PB
ANDNOT 4907.09  ; STACKING LIFTER UPWARD END
LD 4940.02  ; STACKING LIFTER DOWNWARD
AND 4907.10  ; STACKING LIFTER INTERMEDIATE POSITION
AND T1910  ; STACKING CONTAINER
ORLD
OUT 4940.00  ; STACKING HOOK BACKWARD
; rung 67
LD W73.01  ; STACKING HOOK FORWARD
AND 3800.00  ; SURE PUSH BUTTON SWITCH ON
AND 4907.08  ; STACKING LIFTER DOWNWARD END
OUT 4940.01  ; STACKING HOOK FORWARD
; rung 68
LD W73.02  ; STACKING LIFTER DOWNWARD
AND 3800.00  ; SURE PUSH BUTTON SWITCH ON
LD 4940.02  ; STACKING LIFTER DOWNWARD
ANDNOT 4940.03  ; STACKING LIFTER UPWARD
ORLD
OUT 4940.02  ; STACKING LIFTER DOWNWARD

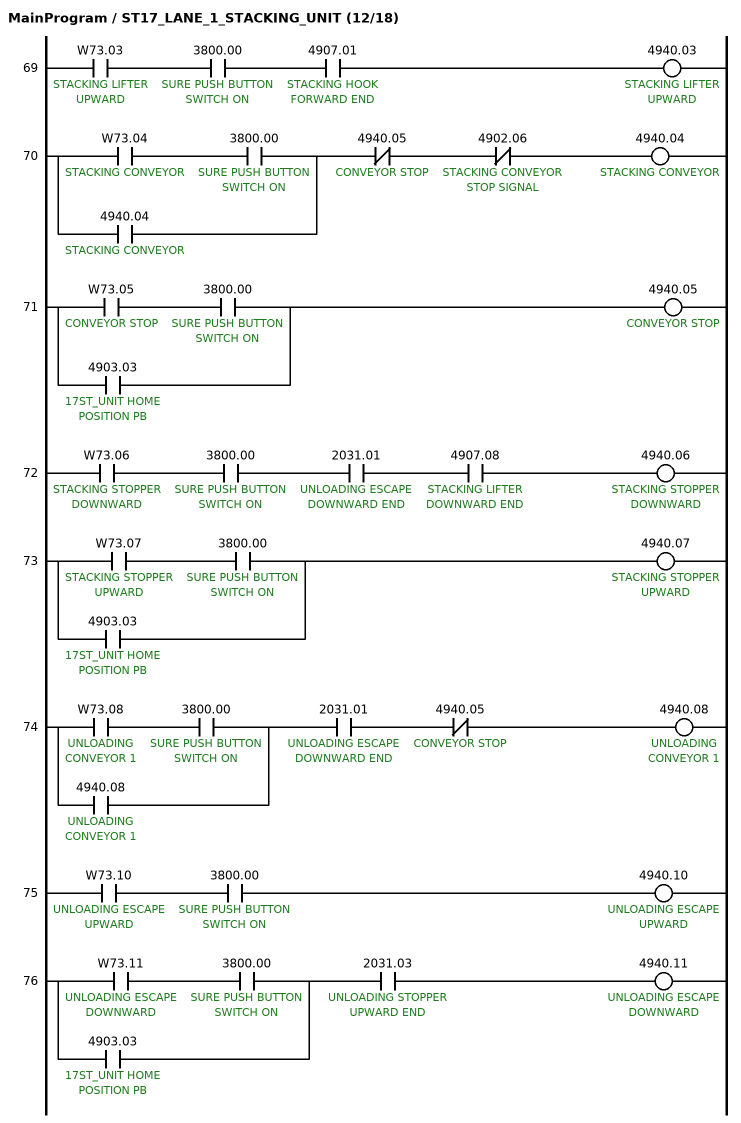
; rung 69
LD W73.03  ; STACKING LIFTER UPWARD
AND 3800.00  ; SURE PUSH BUTTON SWITCH ON
AND 4907.01  ; STACKING HOOK FORWARD END
OUT 4940.03  ; STACKING LIFTER UPWARD
; rung 70
LD W73.04  ; STACKING CONVEYOR
AND 3800.00  ; SURE PUSH BUTTON SWITCH ON
OR 4940.04  ; STACKING CONVEYOR
ANDNOT 4940.05  ; CONVEYOR STOP
ANDNOT 4902.06  ; STACKING CONVEYOR STOP SIGNAL
OUT 4940.04  ; STACKING CONVEYOR
; rung 71
LD W73.05  ; CONVEYOR STOP
AND 3800.00  ; SURE PUSH BUTTON SWITCH ON
OR 4903.03  ; 17ST_UNIT HOME POSITION PB
OUT 4940.05  ; CONVEYOR STOP
; rung 72
LD W73.06  ; STACKING STOPPER DOWNWARD
AND 3800.00  ; SURE PUSH BUTTON SWITCH ON
AND 2031.01  ; UNLOADING ESCAPE DOWNWARD END
AND 4907.08  ; STACKING LIFTER DOWNWARD END
OUT 4940.06  ; STACKING STOPPER DOWNWARD
; rung 73
LD W73.07  ; STACKING STOPPER UPWARD
AND 3800.00  ; SURE PUSH BUTTON SWITCH ON
OR 4903.03  ; 17ST_UNIT HOME POSITION PB
OUT 4940.07  ; STACKING STOPPER UPWARD
; rung 74
LD W73.08  ; UNLOADING CONVEYOR 1
AND 3800.00  ; SURE PUSH BUTTON SWITCH ON
OR 4940.08  ; UNLOADING CONVEYOR 1
AND 2031.01  ; UNLOADING ESCAPE DOWNWARD END
ANDNOT 4940.05  ; CONVEYOR STOP
OUT 4940.08  ; UNLOADING CONVEYOR 1
; rung 75
LD W73.10  ; UNLOADING ESCAPE UPWARD
AND 3800.00  ; SURE PUSH BUTTON SWITCH ON
OUT 4940.10  ; UNLOADING ESCAPE UPWARD
; rung 76
LD W73.11  ; UNLOADING ESCAPE DOWNWARD
AND 3800.00  ; SURE PUSH BUTTON SWITCH ON
OR 4903.03  ; 17ST_UNIT HOME POSITION PB
AND 2031.03  ; UNLOADING STOPPER UPWARD END
OUT 4940.11  ; UNLOADING ESCAPE DOWNWARD

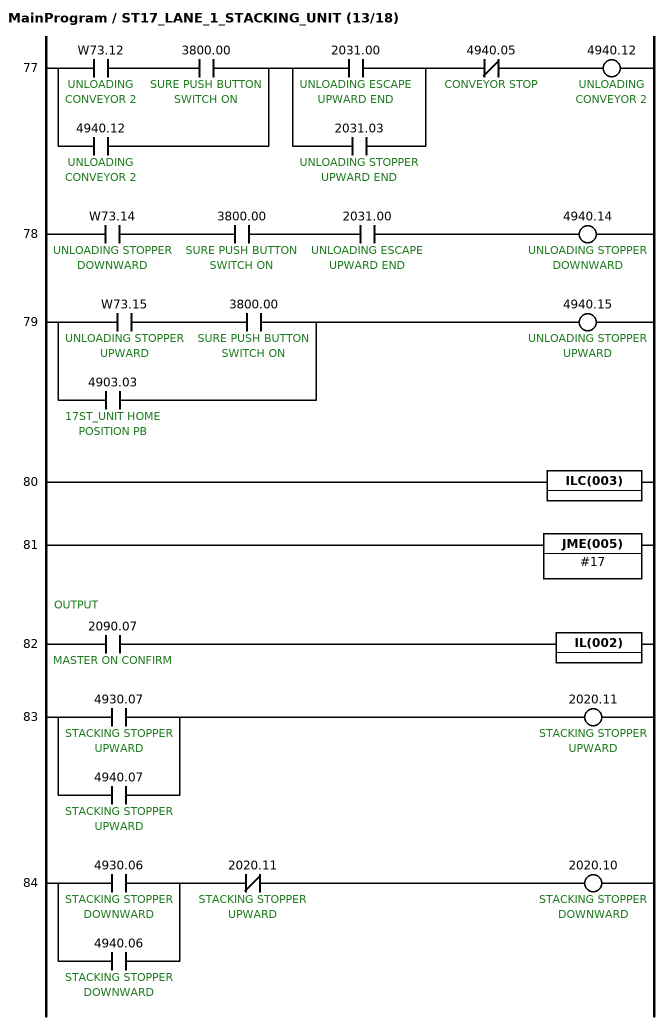
; rung 77
LD W73.12  ; UNLOADING CONVEYOR 2
AND 3800.00  ; SURE PUSH BUTTON SWITCH ON
OR 4940.12  ; UNLOADING CONVEYOR 2
LD 2031.00  ; UNLOADING ESCAPE UPWARD END
OR 2031.03  ; UNLOADING STOPPER UPWARD END
ANDLD
ANDNOT 4940.05  ; CONVEYOR STOP
OUT 4940.12  ; UNLOADING CONVEYOR 2
; rung 78
LD W73.14  ; UNLOADING STOPPER DOWNWARD
AND 3800.00  ; SURE PUSH BUTTON SWITCH ON
AND 2031.00  ; UNLOADING ESCAPE UPWARD END
OUT 4940.14  ; UNLOADING STOPPER DOWNWARD
; rung 79
LD W73.15  ; UNLOADING STOPPER UPWARD
AND 3800.00  ; SURE PUSH BUTTON SWITCH ON
OR 4903.03  ; 17ST_UNIT HOME POSITION PB
OUT 4940.15  ; UNLOADING STOPPER UPWARD
; rung 80
ILC(003)
; rung 81
JME(005) #17
; rung 82: OUTPUT
LD 2090.07  ; MASTER ON CONFIRM
IL(002)
; rung 83
LD 4930.07  ; STACKING STOPPER UPWARD
OR 4940.07  ; STACKING STOPPER UPWARD
OUT 2020.11  ; STACKING STOPPER UPWARD
; rung 84
LD 4930.06  ; STACKING STOPPER DOWNWARD
OR 4940.06  ; STACKING STOPPER DOWNWARD
ANDNOT 2020.11  ; STACKING STOPPER UPWARD
OUT 2020.10  ; STACKING STOPPER DOWNWARD

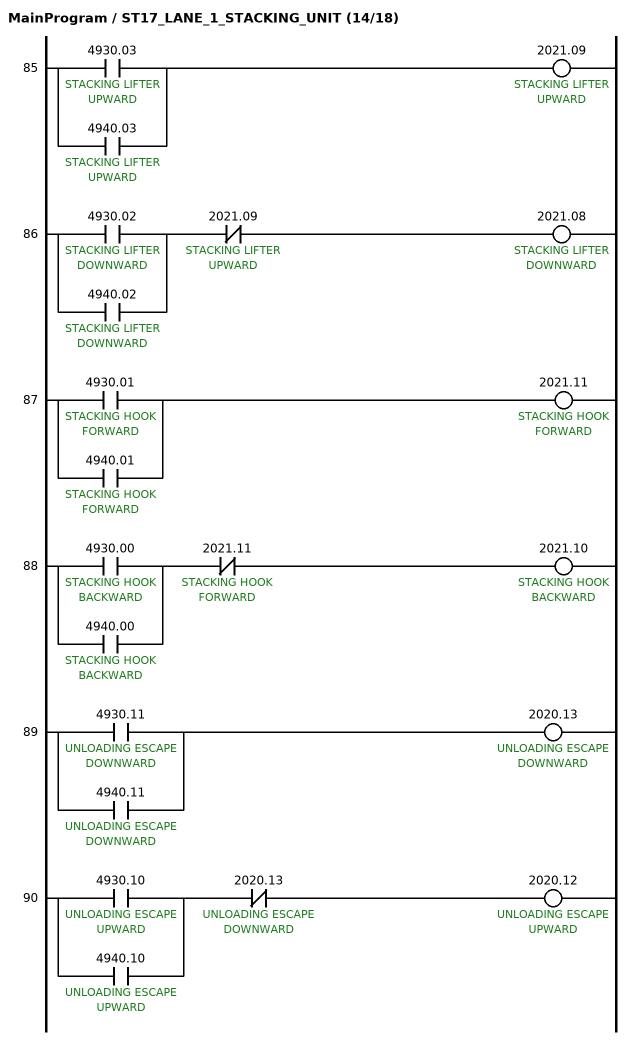
; rung 85
LD 4930.03  ; STACKING LIFTER UPWARD
OR 4940.03  ; STACKING LIFTER UPWARD
OUT 2021.09  ; STACKING LIFTER UPWARD
; rung 86
LD 4930.02  ; STACKING LIFTER DOWNWARD
OR 4940.02  ; STACKING LIFTER DOWNWARD
ANDNOT 2021.09  ; STACKING LIFTER UPWARD
OUT 2021.08  ; STACKING LIFTER DOWNWARD
; rung 87
LD 4930.01  ; STACKING HOOK FORWARD
OR 4940.01  ; STACKING HOOK FORWARD
OUT 2021.11  ; STACKING HOOK FORWARD
; rung 88
LD 4930.00  ; STACKING HOOK BACKWARD
OR 4940.00  ; STACKING HOOK BACKWARD
ANDNOT 2021.11  ; STACKING HOOK FORWARD
OUT 2021.10  ; STACKING HOOK BACKWARD
; rung 89
LD 4930.11  ; UNLOADING ESCAPE DOWNWARD
OR 4940.11  ; UNLOADING ESCAPE DOWNWARD
OUT 2020.13  ; UNLOADING ESCAPE DOWNWARD
; rung 90
LD 4930.10  ; UNLOADING ESCAPE UPWARD
OR 4940.10  ; UNLOADING ESCAPE UPWARD
ANDNOT 2020.13  ; UNLOADING ESCAPE DOWNWARD
OUT 2020.12  ; UNLOADING ESCAPE UPWARD

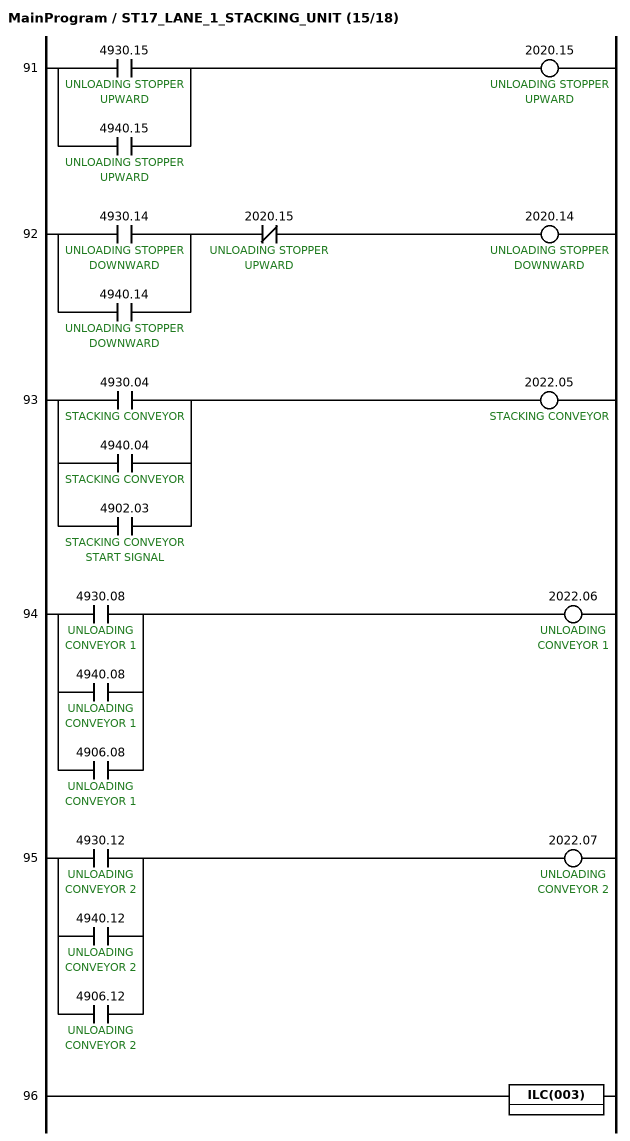
; rung 91
LD 4930.15  ; UNLOADING STOPPER UPWARD
OR 4940.15  ; UNLOADING STOPPER UPWARD
OUT 2020.15  ; UNLOADING STOPPER UPWARD
; rung 92
LD 4930.14  ; UNLOADING STOPPER DOWNWARD
OR 4940.14  ; UNLOADING STOPPER DOWNWARD
ANDNOT 2020.15  ; UNLOADING STOPPER UPWARD
OUT 2020.14  ; UNLOADING STOPPER DOWNWARD
; rung 93
LD 4930.04  ; STACKING CONVEYOR
OR 4940.04  ; STACKING CONVEYOR
OR 4902.03  ; STACKING CONVEYOR START SIGNAL
OUT 2022.05  ; STACKING CONVEYOR
; rung 94
LD 4930.08  ; UNLOADING CONVEYOR 1
OR 4940.08  ; UNLOADING CONVEYOR 1
OR 4906.08  ; UNLOADING CONVEYOR 1
OUT 2022.06  ; UNLOADING CONVEYOR 1
; rung 95
LD 4930.12  ; UNLOADING CONVEYOR 2
OR 4940.12  ; UNLOADING CONVEYOR 2
OR 4906.12  ; UNLOADING CONVEYOR 2
OUT 2022.07  ; UNLOADING CONVEYOR 2
; rung 96
ILC(003)

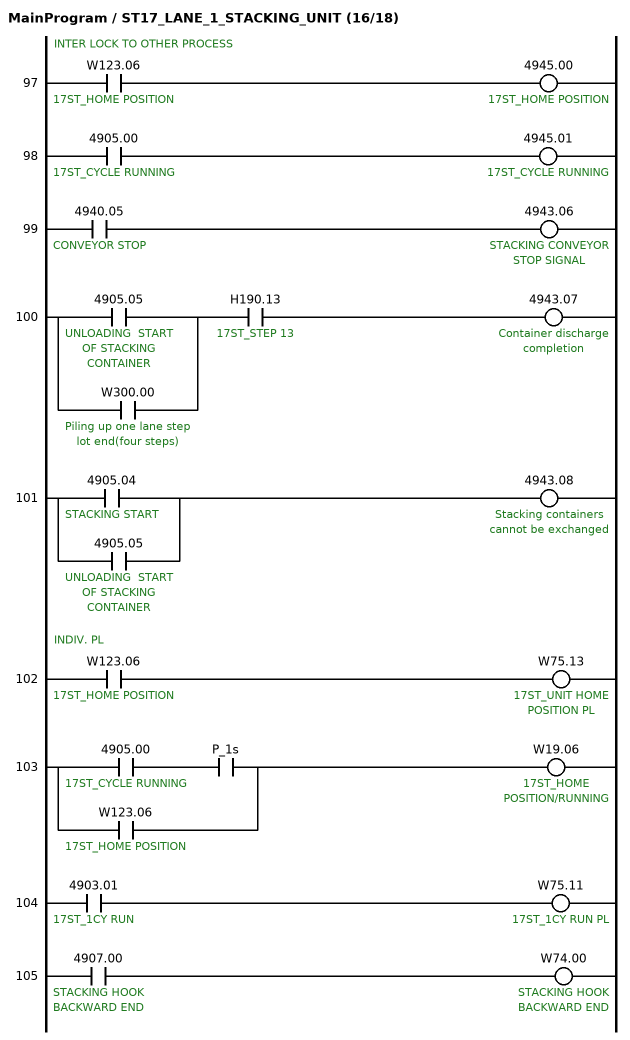
; rung 97: INTER LOCK TO OTHER PROCESS
LD W123.06  ; 17ST_HOME POSITION
OUT 4945.00  ; 17ST_HOME POSITION
; rung 98
LD 4905.00  ; 17ST_CYCLE RUNNING
OUT 4945.01  ; 17ST_CYCLE RUNNING
; rung 99
LD 4940.05  ; CONVEYOR STOP
OUT 4943.06  ; STACKING CONVEYOR STOP SIGNAL
; rung 100
LD 4905.05  ; UNLOADING  START OF STACKING CONTAINER
OR W300.00  ; Piling up one lane step lot end(four steps)
AND H190.13  ; 17ST_STEP 13
OUT 4943.07  ; Container discharge completion
; rung 101
LD 4905.04  ; STACKING START
OR 4905.05  ; UNLOADING  START OF STACKING CONTAINER
OUT 4943.08  ; Stacking containers cannot be exchanged
; rung 102: INDIV. PL
LD W123.06  ; 17ST_HOME POSITION
OUT W75.13  ; 17ST_UNIT HOME POSITION PL
; rung 103
LD 4905.00  ; 17ST_CYCLE RUNNING
AND P_1s
OR W123.06  ; 17ST_HOME POSITION
OUT W19.06  ; 17ST_HOME POSITION/RUNNING
; rung 104
LD 4903.01  ; 17ST_1CY RUN
OUT W75.11  ; 17ST_1CY RUN PL
; rung 105
LD 4907.00  ; STACKING HOOK BACKWARD END
OUT W74.00  ; STACKING HOOK BACKWARD END

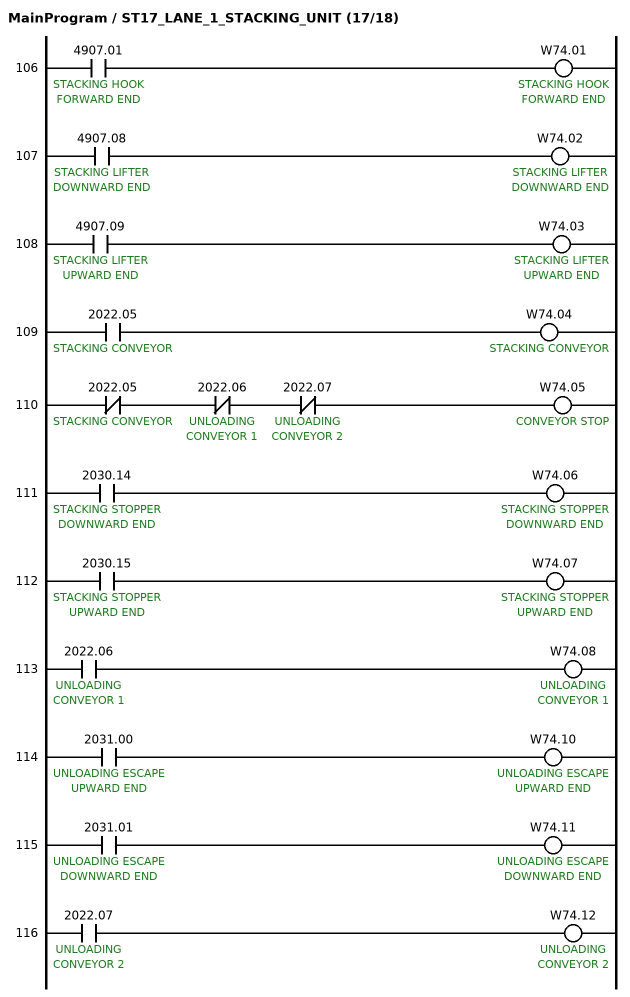
; rung 106
LD 4907.01  ; STACKING HOOK FORWARD END
OUT W74.01  ; STACKING HOOK FORWARD END
; rung 107
LD 4907.08  ; STACKING LIFTER DOWNWARD END
OUT W74.02  ; STACKING LIFTER DOWNWARD END
; rung 108
LD 4907.09  ; STACKING LIFTER UPWARD END
OUT W74.03  ; STACKING LIFTER UPWARD END
; rung 109
LD 2022.05  ; STACKING CONVEYOR
OUT W74.04  ; STACKING CONVEYOR
; rung 110
LDNOT 2022.05  ; STACKING CONVEYOR
ANDNOT 2022.06  ; UNLOADING CONVEYOR 1
ANDNOT 2022.07  ; UNLOADING CONVEYOR 2
OUT W74.05  ; CONVEYOR STOP
; rung 111
LD 2030.14  ; STACKING STOPPER DOWNWARD END
OUT W74.06  ; STACKING STOPPER DOWNWARD END
; rung 112
LD 2030.15  ; STACKING STOPPER UPWARD END
OUT W74.07  ; STACKING STOPPER UPWARD END
; rung 113
LD 2022.06  ; UNLOADING CONVEYOR 1
OUT W74.08  ; UNLOADING CONVEYOR 1
; rung 114
LD 2031.00  ; UNLOADING ESCAPE UPWARD END
OUT W74.10  ; UNLOADING ESCAPE UPWARD END
; rung 115
LD 2031.01  ; UNLOADING ESCAPE DOWNWARD END
OUT W74.11  ; UNLOADING ESCAPE DOWNWARD END
; rung 116
LD 2022.07  ; UNLOADING CONVEYOR 2
OUT W74.12  ; UNLOADING CONVEYOR 2

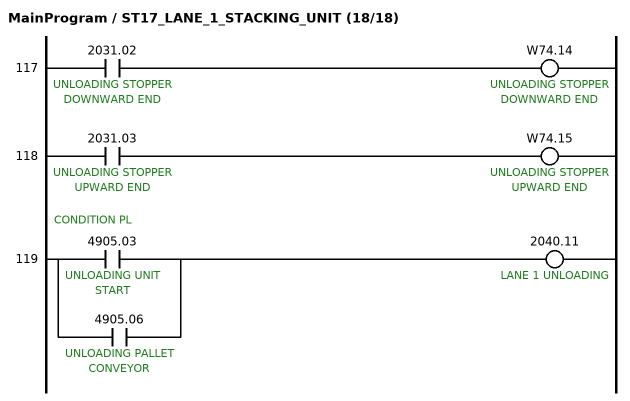
; rung 117
LD 2031.02  ; UNLOADING STOPPER DOWNWARD END
OUT W74.14  ; UNLOADING STOPPER DOWNWARD END
; rung 118
LD 2031.03  ; UNLOADING STOPPER UPWARD END
OUT W74.15  ; UNLOADING STOPPER UPWARD END
; rung 119: CONDITION PL
LD 4905.03  ; UNLOADING UNIT START
OR 4905.06  ; UNLOADING PALLET CONVEYOR
OUT 2040.11  ; LANE 1 UNLOADING

### Section ST18_LANE_2_PALLETIZING_UNIT

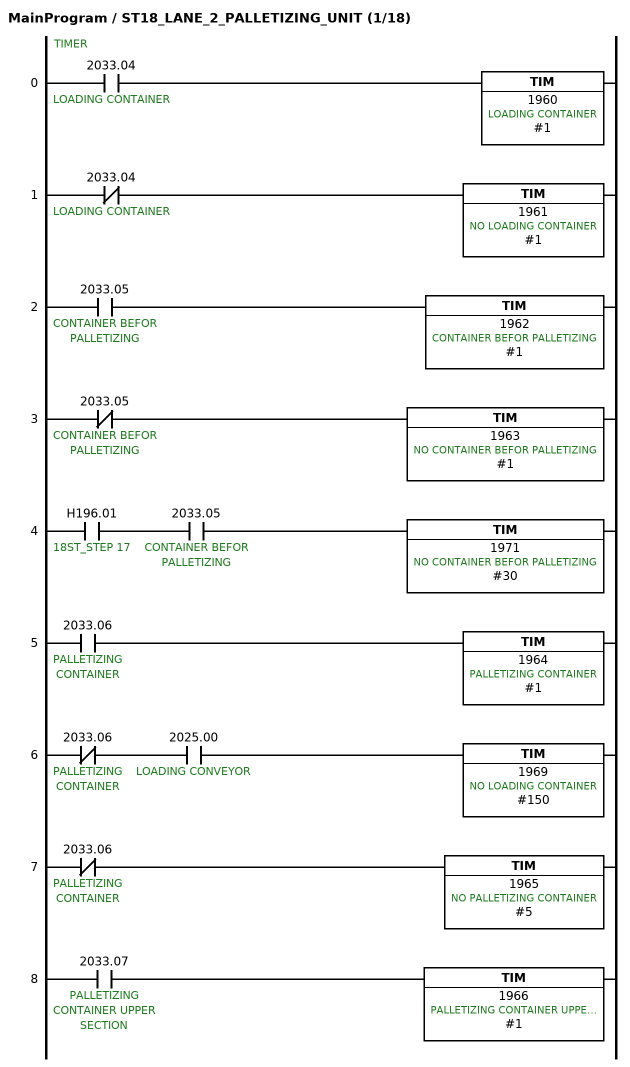
; rung 0: TIMER
LD 2033.04  ; LOADING CONTAINER
TIM 1960 #1  ; LOADING CONTAINER
; rung 1
LDNOT 2033.04  ; LOADING CONTAINER
TIM 1961 #1  ; NO LOADING CONTAINER
; rung 2
LD 2033.05  ; CONTAINER BEFOR PALLETIZING
TIM 1962 #1  ; CONTAINER BEFOR PALLETIZING
; rung 3
LDNOT 2033.05  ; CONTAINER BEFOR PALLETIZING
TIM 1963 #1  ; NO CONTAINER BEFOR PALLETIZING
; rung 4
LD H196.01  ; 18ST_STEP 17
AND 2033.05  ; CONTAINER BEFOR PALLETIZING
TIM 1971 #30  ; NO CONTAINER BEFOR PALLETIZING
; rung 5
LD 2033.06  ; PALLETIZING CONTAINER
TIM 1964 #1  ; PALLETIZING CONTAINER
; rung 6
LDNOT 2033.06  ; PALLETIZING CONTAINER
AND 2025.00  ; LOADING CONVEYOR
TIM 1969 #150  ; NO LOADING CONTAINER
; rung 7
LDNOT 2033.06  ; PALLETIZING CONTAINER
TIM 1965 #5  ; NO PALLETIZING CONTAINER
; rung 8
LD 2033.07  ; PALLETIZING CONTAINER UPPER SECTION
TIM 1966 #1  ; PALLETIZING CONTAINER UPPER SECTION

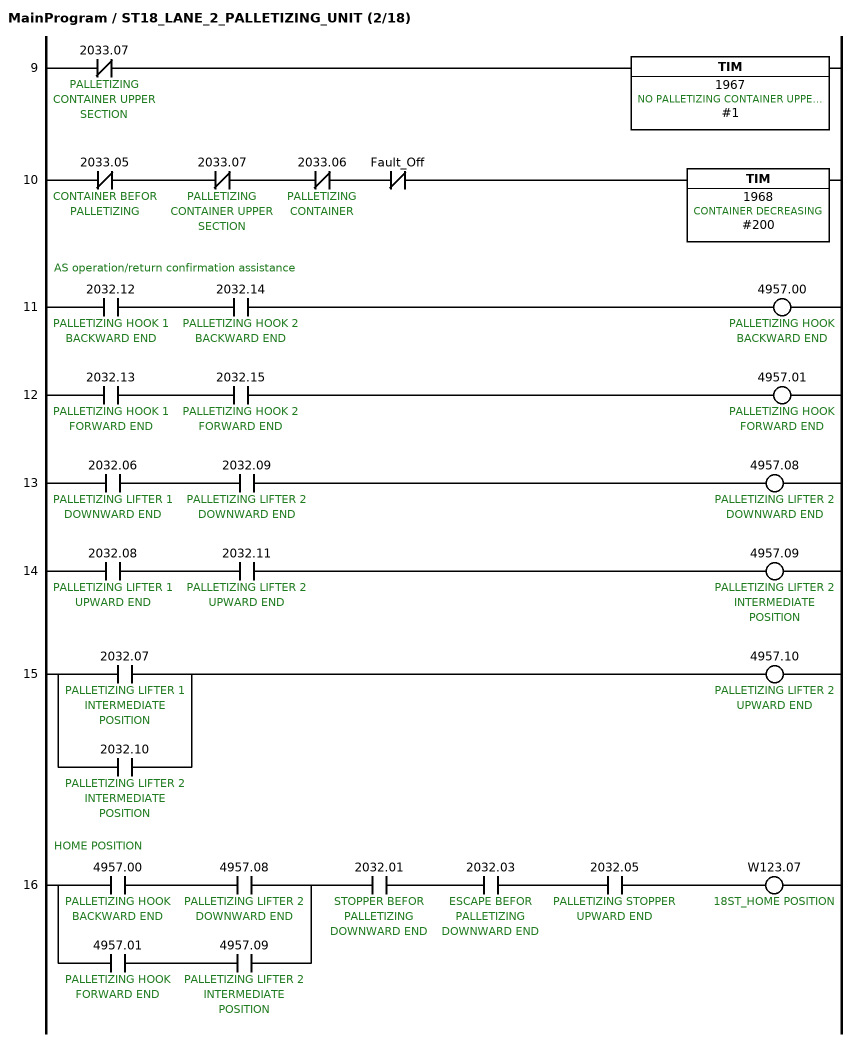
; rung 9
LDNOT 2033.07  ; PALLETIZING CONTAINER UPPER SECTION
TIM 1967 #1  ; NO PALLETIZING CONTAINER UPPER SECTION
; rung 10
LDNOT 2033.05  ; CONTAINER BEFOR PALLETIZING
ANDNOT 2033.07  ; PALLETIZING CONTAINER UPPER SECTION
ANDNOT 2033.06  ; PALLETIZING CONTAINER
ANDNOT Fault_Off
TIM 1968 #200  ; CONTAINER DECREASING
; rung 11: AS operation/return confirmation assistance
LD 2032.12  ; PALLETIZING HOOK 1 BACKWARD END
AND 2032.14  ; PALLETIZING HOOK 2 BACKWARD END
OUT 4957.00  ; PALLETIZING HOOK BACKWARD END
; rung 12
LD 2032.13  ; PALLETIZING HOOK 1 FORWARD END
AND 2032.15  ; PALLETIZING HOOK 2 FORWARD END
OUT 4957.01  ; PALLETIZING HOOK FORWARD END
; rung 13
LD 2032.06  ; PALLETIZING LIFTER 1 DOWNWARD END
AND 2032.09  ; PALLETIZING LIFTER 2 DOWNWARD END
OUT 4957.08  ; PALLETIZING LIFTER 2 DOWNWARD END
; rung 14
LD 2032.08  ; PALLETIZING LIFTER 1 UPWARD END
AND 2032.11  ; PALLETIZING LIFTER 2 UPWARD END
OUT 4957.09  ; PALLETIZING LIFTER 2 INTERMEDIATE POSITION
; rung 15
LD 2032.07  ; PALLETIZING LIFTER 1 INTERMEDIATE POSITION
OR 2032.10  ; PALLETIZING LIFTER 2 INTERMEDIATE POSITION
OUT 4957.10  ; PALLETIZING LIFTER 2 UPWARD END
; rung 16: HOME POSITION
LD 4957.00  ; PALLETIZING HOOK BACKWARD END
AND 4957.08  ; PALLETIZING LIFTER 2 DOWNWARD END
LD 4957.01  ; PALLETIZING HOOK FORWARD END
AND 4957.09  ; PALLETIZING LIFTER 2 INTERMEDIATE POSITION
ORLD
AND 2032.01  ; STOPPER BEFOR PALLETIZING DOWNWARD END
AND 2032.03  ; ESCAPE BEFOR PALLETIZING DOWNWARD END
AND 2032.05  ; PALLETIZING STOPPER UPWARD END
OUT W123.07  ; 18ST_HOME POSITION

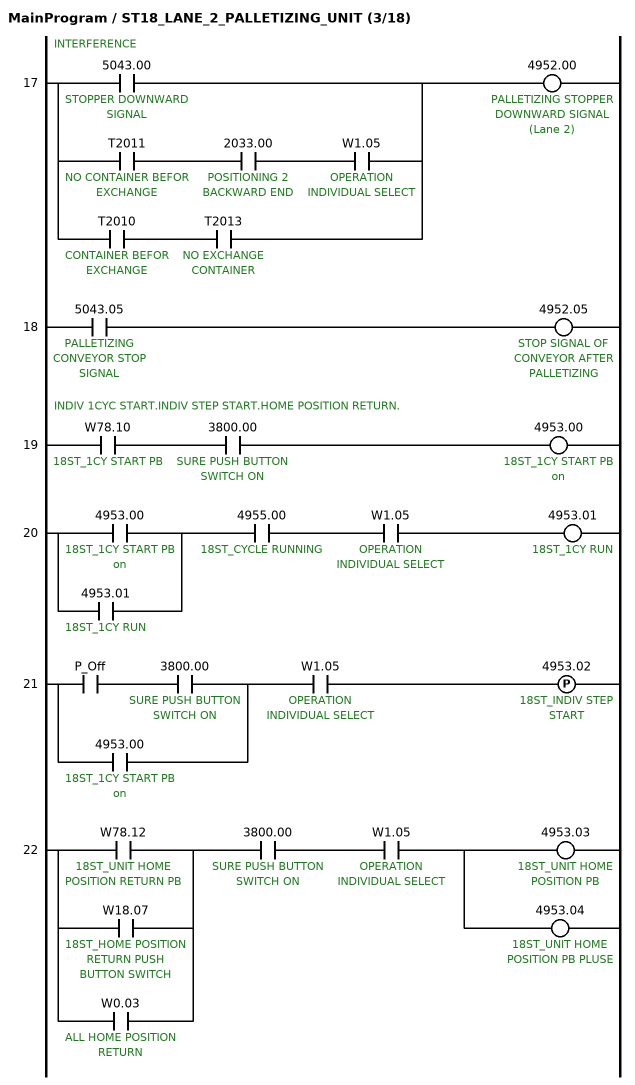
; rung 17: INTERFERENCE
LD 5043.00  ; STOPPER DOWNWARD SIGNAL
LD T2011  ; NO CONTAINER BEFOR EXCHANGE
AND 2033.00  ; POSITIONING 2 BACKWARD END
AND W1.05  ; OPERATION INDIVIDUAL SELECT
ORLD
LD T2010  ; CONTAINER BEFOR EXCHANGE
AND T2013  ; NO EXCHANGE CONTAINER
ORLD
OUT 4952.00  ; PALLETIZING STOPPER DOWNWARD SIGNAL (Lane 2)
; rung 18
LD 5043.05  ; PALLETIZING CONVEYOR STOP SIGNAL
OUT 4952.05  ; STOP SIGNAL OF CONVEYOR AFTER PALLETIZING
; rung 19: INDIV 1CYC START.INDIV STEP START.HOME POSITION RETURN.
LD W78.10  ; 18ST_1CY START PB
AND 3800.00  ; SURE PUSH BUTTON SWITCH ON
OUT 4953.00  ; 18ST_1CY START PB on
; rung 20
LD 4953.00  ; 18ST_1CY START PB on
OR 4953.01  ; 18ST_1CY RUN
AND 4955.00  ; 18ST_CYCLE RUNNING
AND W1.05  ; OPERATION INDIVIDUAL SELECT
OUT 4953.01  ; 18ST_1CY RUN
; rung 21
LD P_Off
AND 3800.00  ; SURE PUSH BUTTON SWITCH ON
OR 4953.00  ; 18ST_1CY START PB on
AND W1.05  ; OPERATION INDIVIDUAL SELECT
DIFU(013) 4953.02  ; 18ST_INDIV STEP START
; rung 22
LD W78.12  ; 18ST_UNIT HOME POSITION RETURN PB
OR W18.07  ; 18ST_HOME POSITION RETURN PUSH BUTTON SWITCH
OR W0.03  ; ALL HOME POSITION RETURN
AND 3800.00  ; SURE PUSH BUTTON SWITCH ON
AND W1.05  ; OPERATION INDIVIDUAL SELECT
OUT 4953.03  ; 18ST_UNIT HOME POSITION PB
OUT 4953.04  ; 18ST_UNIT HOME POSITION PB PLUSE

